FUNCTION_BLOCK V2Q2u
VAR_INPUT
	Ps	: LREAL;
	Pa	: LREAL;
	Pb	: LREAL;
	y	: LREAL;
END_VAR
VAR_OUTPUT
	u		: LREAL;
	Q_lm	: LREAL;
	dP		: LREAL;
END_VAR
VAR
	phi						: LREAL ;
	A						: LREAL ;
	BW 						: LREAL ;
	SpoolTravel 			: LREAL ;
	fSlopeCharacteristic	: LREAL ;
	dpref					: LREAL ;
	dp0						: LREAL ;
	Q						: LREAL ;	
	Q_star					: LREAL ;

END_VAR

phi := 0.7130; 
A := 33.1/10000; 								// Area
BW := 0;										// Bandwidth 
SpoolTravel := 7; 								//Maximum Spool Travel
fSlopeCharacteristic := (SpoolTravel-BW)/25; 	// Valve Slope Characteristic [mm/(L/min)] 
dP0 := 7E5; 									// Pressure drop with compansator 

IF y > 0.0 THEN 
    (* '<S1>:1:11' 
	Q := x_dot * A; *)(* Wanted Flow *)
    (* '<S1>:1:12' 
	dP := (Ps-Pa)*1e5; *)
    
    (* '<S1>:1:13'	
	dp_ref := abs(dP_0/dP); *)
     
    (* '<S1>:1:15' 
	Q_star := (Q * sqrt(dp_ref)) * 6e4; *)
	Q := y * A; // Wanted Flow
	dP := (Ps - Pa) * 100000.0;
    // dpref := ABS(dP0 / dP); 
	dpref := 1;
	
    Q_star := (Q * SQRT(dpref)) * 60000.0;
    (* Outport: '<Root>/u' *)
    (* Referance Flow [L/min] *)
    (* '<S1>:1:16' 
	u := (Q_star * a + BW)/SpoolTravel; *)
    u := (Q_star * (fSlopeCharacteristic+BW)) / SpoolTravel; // Control Signal [-1, 1]
ELSIF y < 0.0 THEN 
    (* '<S1>:1:18' elseif x_dot < 0 *)
    (* '<S1>:1:19' Q := x_dot * (A*phi); *)(* Wanted Flow *)
    (* '<S1>:1:20' dP := (Ps-Pb)*1e5; *)
    dP := (Ps - Pb) * 100000.0;
    (* '<S1>:1:21' dp_ref := abs(dP_0/dP); *)
    (* dp_ref := 1; *)
    (* '<S1>:1:23' Q_star := (Q * sqrt(dp_ref)) * 6e4; *)
    dpref := 1;
	// dpref := ABS(dP0 / dP);
	Q_star := (Q * SQRT(dpref)) * 60000.0;
    (* Outport: '<Root>/u' *)
    (* Referance Flow [L/min] *)
    (* '<S1>:1:24' u := (Q_star * a - BW)/SpoolTravel; *)
	u := (Q_star * (fSlopeCharacteristic - BW)) / SpoolTravel;
    (* Control Signal [-1, 1] *)
ELSE 
    (* '<S1>:1:26' else *)
    (* '<S1>:1:27' Q_star := 0; *)
    Q_star := 0.0;
    (* '<S1>:1:28' dP := 0; *)
    dP := 0.0;
    (* Outport: '<Root>/u' *)
    (* '<S1>:1:29' u := 0; *)
    u := 0.0;
END_IF;

(* Outport: '<Root>/Q_lm' incorporates:
 *  MATLAB Function: '<Root>/V2Q2u' *)
(* '<S1>:1:32' Q_lm := Q_star; *)
(* Q * 6E4; *)
Q_lm := Q_star;

END_FUNCTION_BLOCK

(* stored: Version 1.1.0.1, ProductVersion 3.1.4024.13
   POU V2Q2u: Id {8efb5770-48c6-4830-a612-83b6696c3542}, SpecialFunc None *)
